// Empty function block that extends an empty function block.
FUNCTION_BLOCK FB_EmptyWithExtends EXTENDS FB_Empty
VAR
END_VAR

END_FUNCTION_BLOCK

(* stored: Version 1.1.0.1, ProductVersion 3.1.4024.15
   POU FB_EmptyWithExtends: Id {80774b89-1675-49f7-aa30-1aa04710438c}, SpecialFunc None *)
